FUNCTION_BLOCK SpeedSimulation (* Basic Function Block Type *)
  (* Standard: 61499-2 *)
  (* Version 0.0, 6/12/2026, Schneider Electric, Template *)
  PACKAGE SE.Nereda;
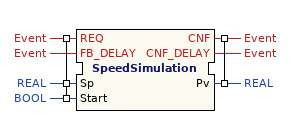
  EVENT_INPUT
    REQ WITH Sp, Start; (* Normal Execution Request *)
    FB_DELAY;
  END_EVENT
  EVENT_OUTPUT
    CNF WITH Pv; (* Execution Confirmation *)
    CNF_DELAY;
  END_EVENT
  VAR_INPUT
    Sp : REAL; (* Input event qualifier *)
    Start : BOOL;
  END_VAR
  VAR_OUTPUT
    Pv : REAL; (* Output event qualifier *)
  END_VAR
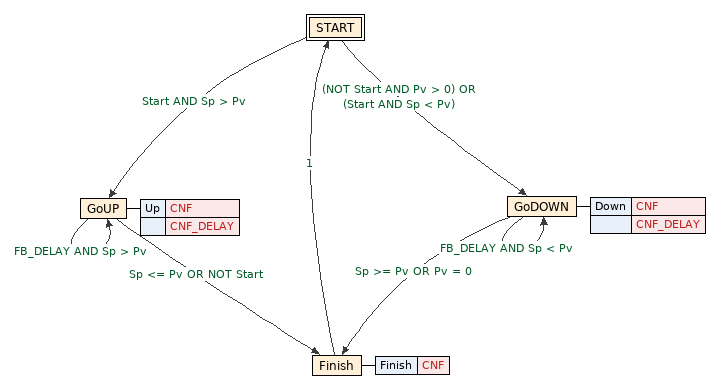
  EC_STATES
    START; (* Initial State *)
    GoUP : Up -> CNF, -> CNF_DELAY;
    GoDOWN : Down -> CNF, -> CNF_DELAY;
    Finish : Finish -> CNF;
  END_STATES
  EC_TRANSITIONS
    START TO GoUP := Start AND Sp > Pv;
    START TO GoDOWN := (NOT Start AND Pv > 0) OR (Start AND Sp < Pv);
    GoDOWN TO GoDOWN := FB_DELAY AND Sp < Pv;
    GoUP TO GoUP := FB_DELAY AND Sp > Pv;
    GoDOWN TO Finish := Sp >= Pv OR Pv = 0;
    GoUP TO Finish := Sp <= Pv OR NOT Start;
    Finish TO START := 1;
  END_TRANSITIONS
  ALGORITHM Up IN ST:
;
Pv := Pv + 1;
  END_ALGORITHM
  ALGORITHM Down IN ST:
;
Pv := Pv - 1;
  END_ALGORITHM
  ALGORITHM Finish IN ST:
;
IF Pv < 0 THEN
	Pv := 0;
ELSIF Start THEN
	Pv := Sp;
END_IF;
  END_ALGORITHM
END_FUNCTION_BLOCK
